// TIA Portal V16 export
// export: Created 2024-06-24T15:42:27.5574986Z, ExportSetting WithDefaults, DisplayName Totally Integrated Automation Portal, DisplayVersion V16, DisplayName TIA Portal Version Control Interface, DisplayVersion V16, DisplayName TIA Portal Openness, DisplayVersion V16, DisplayName STEP 7 Professional, DisplayVersion V16, DisplayName STEP 7 Safety, DisplayVersion V16, DisplayName WinCC Advanced, DisplayVersion V16
FUNCTION_BLOCK "FB_Main"   // FB2, LAD
{ S7_Optimized_Access := 'TRUE' }
VERSION : 0.1
// stored: AutoNumber true, IsIECCheckEnabled false, IsRetainMemResEnabled false, MemoryReserve 100, SetENOAutomatically false, UDAEnableTagReadback false
   VAR
      FB_Conveyor_Entry { S7_SetPoint := 'True'} : "FB_Conveyor";
      FB_Conveyor_Weight { S7_SetPoint := 'True'} : "FB_Conveyor";
      FB_WheelSorter_Instance { S7_SetPoint := 'True'} : "FB_WheelSorter";
      FB_Conveyor_Left { S7_SetPoint := 'True'} : "FB_Conveyor";
      FB_Conveyor_Straight { S7_SetPoint := 'True'} : "FB_Conveyor";
      FB_Conveyor_Right { S7_SetPoint := 'True'} : "FB_Conveyor";
      FB_PickAndPlace_Instance { S7_SetPoint := 'True'} : "FB_PickAndPlace";
      FB_Conveyor_4belt { S7_SetPoint := 'True'} : "FB_Conveyor";
   END_VAR
BEGIN

REGION Network 1
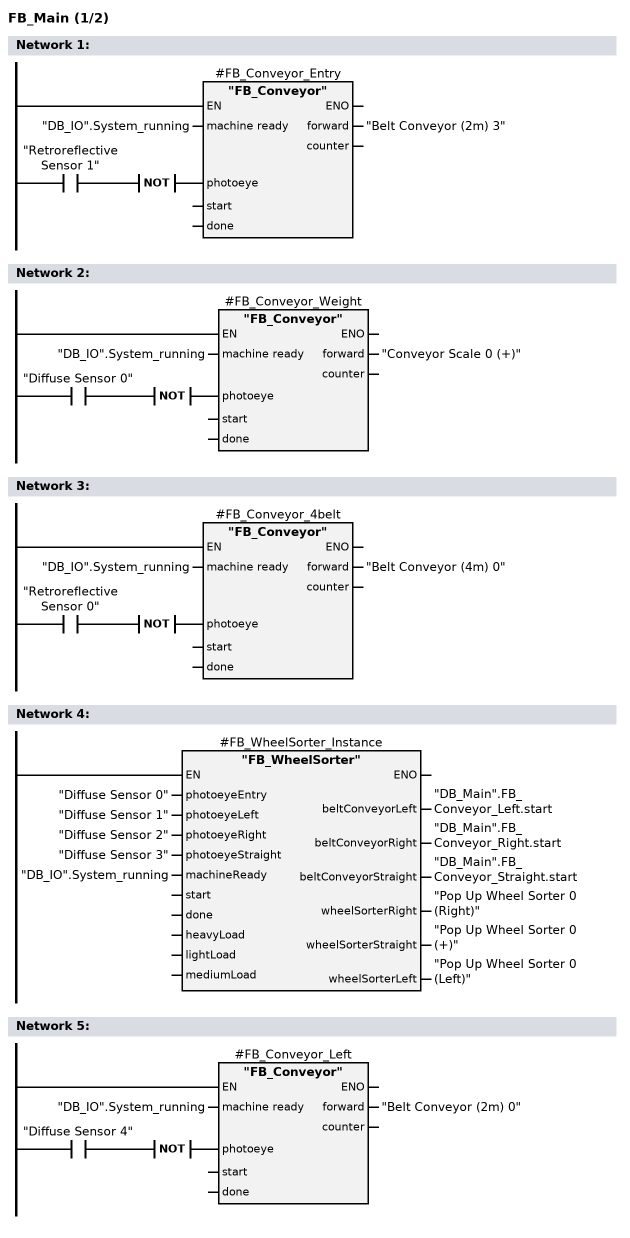
   RUNG wire#powerrail
      #FB_Conveyor_Entry(photoeye := wire#w1, "machine ready" := "DB_IO".System_running, start :=, done :=, forward => "Belt Conveyor (2m) 3", "counter" =>)
   END_RUNG
   RUNG wire#powerrail
      Contact( "Retroreflective Sensor 1" )
      Not()
   END_RUNG wire#w1
   // the same network as SCL:
   #FB_Conveyor_Entry("machine ready" := "DB_IO".System_running,   // "FB_Conveyor"
                      photoeye := NOT "Retroreflective Sensor 1",
                      forward => "Belt Conveyor (2m) 3");
END_REGION

REGION Network 2
   RUNG wire#powerrail
      #FB_Conveyor_Weight(photoeye := wire#w1, "machine ready" := "DB_IO".System_running, start :=, done :=, forward => "Conveyor Scale 0 (+)", "counter" =>)
   END_RUNG
   RUNG wire#powerrail
      Contact( "Diffuse Sensor 0" )
      Not()
   END_RUNG wire#w1
   // the same network as SCL:
   #FB_Conveyor_Weight("machine ready" := "DB_IO".System_running,   // "FB_Conveyor"
                       photoeye := NOT "Diffuse Sensor 0",
                       forward => "Conveyor Scale 0 (+)");
END_REGION

REGION Network 3
   RUNG wire#powerrail
      #FB_Conveyor_4belt(photoeye := wire#w1, "machine ready" := "DB_IO".System_running, start :=, done :=, forward => "Belt Conveyor (4m) 0", "counter" =>)
   END_RUNG
   RUNG wire#powerrail
      Contact( "Retroreflective Sensor 0" )
      Not()
   END_RUNG wire#w1
   // the same network as SCL:
   #FB_Conveyor_4belt("machine ready" := "DB_IO".System_running,   // "FB_Conveyor"
                      photoeye := NOT "Retroreflective Sensor 0",
                      forward => "Belt Conveyor (4m) 0");
END_REGION

REGION Network 4
   RUNG wire#powerrail
      #FB_WheelSorter_Instance(photoeyeEntry := "Diffuse Sensor 0", photoeyeLeft := "Diffuse Sensor 1", photoeyeRight := "Diffuse Sensor 2", photoeyeStraight := "Diffuse Sensor 3", machineReady := "DB_IO".System_running, start :=, done :=, heavyLoad :=, lightLoad :=, mediumLoad :=, beltConveyorLeft => "DB_Main".FB_Conveyor_Left.start, beltConveyorRight => "DB_Main".FB_Conveyor_Right.start, beltConveyorStraight => "DB_Main".FB_Conveyor_Straight.start, wheelSorterRight => "Pop Up Wheel Sorter 0 (Right)", wheelSorterStraight => "Pop Up Wheel Sorter 0 (+)", wheelSorterLeft => "Pop Up Wheel Sorter 0 (Left)")
   END_RUNG
   // the same network as SCL:
   #FB_WheelSorter_Instance(photoeyeEntry := "Diffuse Sensor 0",   // "FB_WheelSorter"
                           photoeyeLeft := "Diffuse Sensor 1",
                           photoeyeRight := "Diffuse Sensor 2",
                           photoeyeStraight := "Diffuse Sensor 3",
                           machineReady := "DB_IO".System_running,
                           beltConveyorLeft => "DB_Main".FB_Conveyor_Left.start,
                           beltConveyorRight => "DB_Main".FB_Conveyor_Right.start,
                           beltConveyorStraight => "DB_Main".FB_Conveyor_Straight.start,
                           wheelSorterRight => "Pop Up Wheel Sorter 0 (Right)",
                           wheelSorterStraight => "Pop Up Wheel Sorter 0 (+)",
                           wheelSorterLeft => "Pop Up Wheel Sorter 0 (Left)");
END_REGION

REGION Network 5
   RUNG wire#powerrail
      #FB_Conveyor_Left(photoeye := wire#w1, "machine ready" := "DB_IO".System_running, start :=, done :=, forward => "Belt Conveyor (2m) 0", "counter" =>)
   END_RUNG
   RUNG wire#powerrail
      Contact( "Diffuse Sensor 4" )
      Not()
   END_RUNG wire#w1
   // the same network as SCL:
   #FB_Conveyor_Left("machine ready" := "DB_IO".System_running,   // "FB_Conveyor"
                     photoeye := NOT "Diffuse Sensor 4",
                     forward => "Belt Conveyor (2m) 0");
END_REGION

REGION Network 6
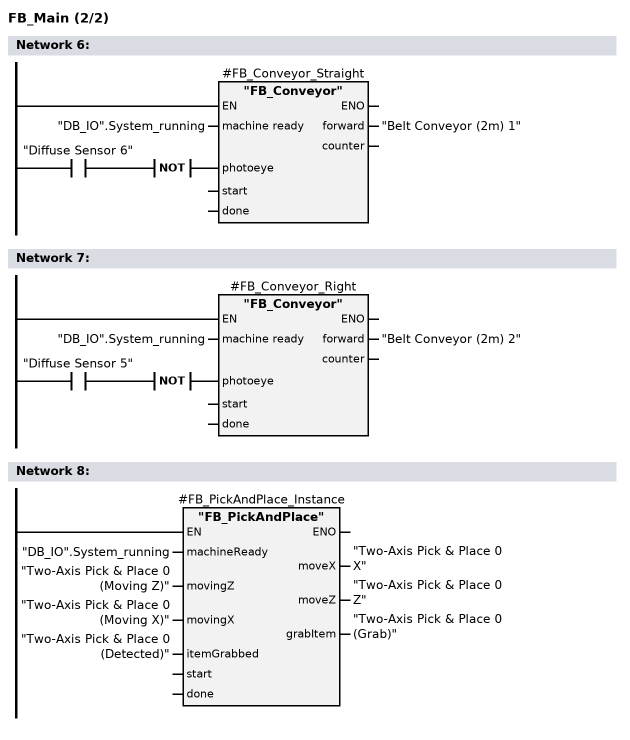
   RUNG wire#powerrail
      #FB_Conveyor_Straight(photoeye := wire#w1, "machine ready" := "DB_IO".System_running, start :=, done :=, forward => "Belt Conveyor (2m) 1", "counter" =>)
   END_RUNG
   RUNG wire#powerrail
      Contact( "Diffuse Sensor 6" )
      Not()
   END_RUNG wire#w1
   // the same network as SCL:
   #FB_Conveyor_Straight("machine ready" := "DB_IO".System_running,   // "FB_Conveyor"
                         photoeye := NOT "Diffuse Sensor 6",
                         forward => "Belt Conveyor (2m) 1");
END_REGION

REGION Network 7
   RUNG wire#powerrail
      #FB_Conveyor_Right(photoeye := wire#w1, "machine ready" := "DB_IO".System_running, start :=, done :=, forward => "Belt Conveyor (2m) 2", "counter" =>)
   END_RUNG
   RUNG wire#powerrail
      Contact( "Diffuse Sensor 5" )
      Not()
   END_RUNG wire#w1
   // the same network as SCL:
   #FB_Conveyor_Right("machine ready" := "DB_IO".System_running,   // "FB_Conveyor"
                      photoeye := NOT "Diffuse Sensor 5",
                      forward => "Belt Conveyor (2m) 2");
END_REGION

REGION Network 8
   #FB_PickAndPlace_Instance(machineReady := "DB_IO".System_running,   // "FB_PickAndPlace"
                           movingZ := "Two-Axis Pick & Place 0 (Moving Z)",
                           movingX := "Two-Axis Pick & Place 0 (Moving X)",
                           itemGrabbed := "Two-Axis Pick & Place 0 (Detected)",
                           moveX => "Two-Axis Pick & Place 0 X",
                           moveZ => "Two-Axis Pick & Place 0 Z",
                           grabItem => "Two-Axis Pick & Place 0 (Grab)");
END_REGION
END_FUNCTION_BLOCK
